DATA_BLOCK "FM350_DB"
TITLE =
VERSION : 0.1

 UDT 1
BEGIN
   JOB_WR.NO := B#16#0;
   JOB_WR.BUSY := FALSE;
   JOB_WR.DONE := FALSE;
   JOB_WR.IMPOSS := FALSE;
   JOB_WR.UNKOWN := FALSE;
   JOB_RD.NO := B#16#0;
   JOB_RD.BUSY := FALSE;
   JOB_RD.DONE := FALSE;
   JOB_RD.IMPOSS := FALSE;
   JOB_RD.UNKOWN := FALSE;
   RESERV_0[1] := W#16#0;
   RESERV_0[2] := W#16#0;
   RESERV_0[3] := W#16#0;
   RESERV_1 := W#16#0;
   MOD_ADR := W#16#100;
   CH_ADR := DW#16#800;
   DS_OFFS := B#16#0;
   RESERV_2 := B#16#0;
   CONTROL_SIGNALS.BIT0_0 := FALSE;
   CONTROL_SIGNALS.BIT0_1 := FALSE;
   CONTROL_SIGNALS.BIT0_2 := FALSE;
   CONTROL_SIGNALS.BIT0_3 := FALSE;
   CONTROL_SIGNALS.BIT0_4 := FALSE;
   CONTROL_SIGNALS.BIT0_5 := FALSE;
   CONTROL_SIGNALS.BIT0_6 := FALSE;
   CONTROL_SIGNALS.BIT0_7 := FALSE;
   CONTROL_SIGNALS.CTRL_DQ0 := FALSE;
   CONTROL_SIGNALS.CTRL_DQ1 := FALSE;
   CONTROL_SIGNALS.CTRL_DQ2 := FALSE;
   CONTROL_SIGNALS.CTRL_DQ3 := FALSE;
   CONTROL_SIGNALS.CTRL_DQ4 := FALSE;
   CONTROL_SIGNALS.CTRL_DQ5 := FALSE;
   CONTROL_SIGNALS.CTRL_DQ6 := FALSE;
   CONTROL_SIGNALS.CTRL_DQ7 := FALSE;
   CONTROL_SIGNALS.SET_DQ0 := FALSE;
   CONTROL_SIGNALS.SET_DQ1 := FALSE;
   CONTROL_SIGNALS.SET_DQ2 := FALSE;
   CONTROL_SIGNALS.SET_DQ3 := FALSE;
   CONTROL_SIGNALS.SET_DQ4 := FALSE;
   CONTROL_SIGNALS.SET_DQ5 := FALSE;
   CONTROL_SIGNALS.SET_DQ6 := FALSE;
   CONTROL_SIGNALS.SET_DQ7 := FALSE;
   CONTROL_SIGNALS.SW_GATE0 := FALSE;
   CONTROL_SIGNALS.SW_GATE1 := FALSE;
   CONTROL_SIGNALS.SW_GATE2 := FALSE;
   CONTROL_SIGNALS.SW_GATE3 := FALSE;
   CONTROL_SIGNALS.SW_GATE4 := FALSE;
   CONTROL_SIGNALS.SW_GATE5 := FALSE;
   CONTROL_SIGNALS.SW_GATE6 := FALSE;
   CONTROL_SIGNALS.SW_GATE7 := FALSE;
   CONTROL_SIGNALS.CTRL_DWORD1 := DW#16#0;
   CONTROL_SIGNALS.CTRL_DWORD2 := DW#16#0;
   CONTROL_SIGNALS.CTRL_DWORD3 := DW#16#0;
   CHECKBACK_SIGNALS.BIT0_0 := FALSE;
   CHECKBACK_SIGNALS.STS_TFB := FALSE;
   CHECKBACK_SIGNALS.BIT0_2 := FALSE;
   CHECKBACK_SIGNALS.BIT0_3 := FALSE;
   CHECKBACK_SIGNALS.DATA_ERR := FALSE;
   CHECKBACK_SIGNALS.BIT0_5 := FALSE;
   CHECKBACK_SIGNALS.BIT0_6 := FALSE;
   CHECKBACK_SIGNALS.PARA := FALSE;
   CHECKBACK_SIGNALS.STS_CMP0 := FALSE;
   CHECKBACK_SIGNALS.STS_CMP1 := FALSE;
   CHECKBACK_SIGNALS.STS_CMP2 := FALSE;
   CHECKBACK_SIGNALS.STS_CMP3 := FALSE;
   CHECKBACK_SIGNALS.STS_CMP4 := FALSE;
   CHECKBACK_SIGNALS.STS_CMP5 := FALSE;
   CHECKBACK_SIGNALS.STS_CMP6 := FALSE;
   CHECKBACK_SIGNALS.STS_CMP7 := FALSE;
   CHECKBACK_SIGNALS.STS_UFLW0 := FALSE;
   CHECKBACK_SIGNALS.STS_UFLW1 := FALSE;
   CHECKBACK_SIGNALS.STS_UFLW2 := FALSE;
   CHECKBACK_SIGNALS.STS_UFLW3 := FALSE;
   CHECKBACK_SIGNALS.STS_UFLW4 := FALSE;
   CHECKBACK_SIGNALS.STS_UFLW5 := FALSE;
   CHECKBACK_SIGNALS.STS_UFLW6 := FALSE;
   CHECKBACK_SIGNALS.STS_UFLW7 := FALSE;
   CHECKBACK_SIGNALS.STS_OFLW0 := FALSE;
   CHECKBACK_SIGNALS.STS_OFLW1 := FALSE;
   CHECKBACK_SIGNALS.STS_OFLW2 := FALSE;
   CHECKBACK_SIGNALS.STS_OFLW3 := FALSE;
   CHECKBACK_SIGNALS.STS_OFLW4 := FALSE;
   CHECKBACK_SIGNALS.STS_OFLW5 := FALSE;
   CHECKBACK_SIGNALS.STS_OFLW6 := FALSE;
   CHECKBACK_SIGNALS.STS_OFLW7 := FALSE;
   CHECKBACK_SIGNALS.STS_DIR0 := FALSE;
   CHECKBACK_SIGNALS.STS_DIR1 := FALSE;
   CHECKBACK_SIGNALS.STS_DIR2 := FALSE;
   CHECKBACK_SIGNALS.STS_DIR3 := FALSE;
   CHECKBACK_SIGNALS.STS_DIR4 := FALSE;
   CHECKBACK_SIGNALS.STS_DIR5 := FALSE;
   CHECKBACK_SIGNALS.STS_DIR6 := FALSE;
   CHECKBACK_SIGNALS.STS_DIR7 := FALSE;
   CHECKBACK_SIGNALS.STS_DI0 := FALSE;
   CHECKBACK_SIGNALS.STS_DI1 := FALSE;
   CHECKBACK_SIGNALS.STS_DI2 := FALSE;
   CHECKBACK_SIGNALS.STS_DI3 := FALSE;
   CHECKBACK_SIGNALS.STS_DI4 := FALSE;
   CHECKBACK_SIGNALS.STS_DI5 := FALSE;
   CHECKBACK_SIGNALS.STS_DI6 := FALSE;
   CHECKBACK_SIGNALS.STS_DI7 := FALSE;
   CHECKBACK_SIGNALS.STS_DQ0 := FALSE;
   CHECKBACK_SIGNALS.STS_DQ1 := FALSE;
   CHECKBACK_SIGNALS.STS_DQ2 := FALSE;
   CHECKBACK_SIGNALS.STS_DQ3 := FALSE;
   CHECKBACK_SIGNALS.STS_DQ4 := FALSE;
   CHECKBACK_SIGNALS.STS_DQ5 := FALSE;
   CHECKBACK_SIGNALS.STS_DQ6 := FALSE;
   CHECKBACK_SIGNALS.STS_DQ7 := FALSE;
   CHECKBACK_SIGNALS.STS_GATE0 := FALSE;
   CHECKBACK_SIGNALS.STS_GATE1 := FALSE;
   CHECKBACK_SIGNALS.STS_GATE2 := FALSE;
   CHECKBACK_SIGNALS.STS_GATE3 := FALSE;
   CHECKBACK_SIGNALS.STS_GATE4 := FALSE;
   CHECKBACK_SIGNALS.STS_GATE5 := FALSE;
   CHECKBACK_SIGNALS.STS_GATE6 := FALSE;
   CHECKBACK_SIGNALS.STS_GATE7 := FALSE;
   CHECKBACK_SIGNALS.USER_STAT_WORD0 := W#16#0;
   CHECKBACK_SIGNALS.USER_STAT_WORD1 := W#16#0;
   CHECKBACK_SIGNALS.USER_STAT_WORD2 := W#16#0;
   CHECKBACK_SIGNALS.USER_STAT_WORD3 := W#16#0;
   LOAD_VAL0 := L#0;
   LOAD_VAL1 := L#0;
   LOAD_VAL2 := L#0;
   LOAD_VAL3 := L#0;
   LOAD_VAL4 := L#0;
   LOAD_VAL5 := L#0;
   LOAD_VAL6 := L#0;
   LOAD_VAL7 := L#0;
   LOAD_PREPARE_VAL0 := L#0;
   LOAD_PREPARE_VAL1 := L#0;
   LOAD_PREPARE_VAL2 := L#0;
   LOAD_PREPARE_VAL3 := L#0;
   LOAD_PREPARE_VAL4 := L#0;
   LOAD_PREPARE_VAL5 := L#0;
   LOAD_PREPARE_VAL6 := L#0;
   LOAD_PREPARE_VAL7 := L#0;
   CMP_VAL0 := L#0;
   CMP_VAL1 := L#0;
   CMP_VAL2 := L#0;
   CMP_VAL3 := L#0;
   CMP_VAL4 := L#0;
   CMP_VAL5 := L#0;
   CMP_VAL6 := L#0;
   CMP_VAL7 := L#0;
   ACT_CNTV0 := L#0;
   ACT_MSRV0 := L#0;
   ACT_CNTV1 := L#0;
   ACT_MSRV1 := L#0;
   ACT_CNTV2 := L#0;
   ACT_MSRV2 := L#0;
   ACT_CNTV3 := L#0;
   ACT_MSRV3 := L#0;
   ACT_CNTV4 := L#0;
   ACT_MSRV4 := L#0;
   ACT_CNTV5 := L#0;
   ACT_MSRV5 := L#0;
   ACT_CNTV6 := L#0;
   ACT_MSRV6 := L#0;
   ACT_CNTV7 := L#0;
   ACT_MSRV7 := L#0;
   DIAGNOSTIC_INT_INFO.BYTE0 := B#16#0;
   DIAGNOSTIC_INT_INFO.BYTE1 := B#16#0;
   DIAGNOSTIC_INT_INFO.BYTE2 := B#16#0;
   DIAGNOSTIC_INT_INFO.BYTE3 := B#16#0;
   DIAGNOSTIC_INT_INFO.BYTE4 := B#16#0;
   DIAGNOSTIC_INT_INFO.BYTE5 := B#16#0;
   DIAGNOSTIC_INT_INFO.BYTE6 := B#16#0;
   DIAGNOSTIC_INT_INFO.BYTE7 := B#16#0;
   DIAGNOSTIC_INT_INFO.BYTE8 := B#16#0;
   DIAGNOSTIC_INT_INFO.BYTE9 := B#16#0;
   DIAGNOSTIC_INT_INFO.BYTE10 := B#16#0;
   DIAGNOSTIC_INT_INFO.BYTE11 := B#16#0;
   DIAGNOSTIC_INT_INFO.BYTE12 := B#16#0;
   DIAGNOSTIC_INT_INFO.BYTE13 := B#16#0;
   DIAGNOSTIC_INT_INFO.BYTE14 := B#16#0;
   DIAGNOSTIC_INT_INFO.BYTE15 := B#16#0;
END_DATA_BLOCK

